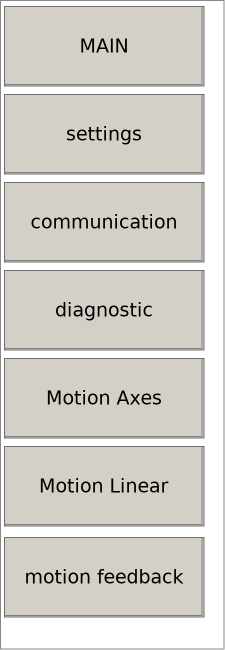
VISUALIZATION MenuMain  // 225x650
    Button (4,94 200x80), "settings"
        OnMouseClick: change screen: APP_Settings
    Button (4,182 200x80), "communication"
        OnMouseClick: change screen: communication
    Button (4,358 200x80), "Motion Axes"
        OnMouseClick: change screen: Motion_Axes
    Button (4,537 200x80), "motion feedback"
        OnMouseClick: change screen: Motion_FBK
    Button (4,6 200x80), "MAIN"
        OnMouseClick: change screen: MainScreen
    Button (4,446 200x80), "Motion Linear"
        OnMouseClick: change screen: Motion_Linear
    Button (4,270 200x80), "diagnostic"
        OnMouseClick: change screen: diagnostic
END_VISUALIZATION

(* stored: Version 1.1.0.1, ProductVersion 3.1.4024.10
   Visu MenuMain: Id {53cc7cd1-366d-4b3b-ad37-5f33e92ed827} *)
